ABB RobotStudio station: IRB_910SC.rsstnx

Station IRB_910SC (saved by RobotStudio 25.5.11605.0)
Controller IRB910SC_3_45
  mechanical unit ROB_1: IRB910SC_3_45__01, 4 joints, base frame (0, 0, 0) mm
Layout (positions relative to the parent item):
  - IRB910SC_3_45__01 [mechanism, from %ABB.RobotStudio.Models.IRB910SC%\IRB910SC_3_45__01.rslib] at (0, 0, 0) mm; joint values [0, 0, 0, 0] (rad or m)
